FUNCTION_BLOCK FB_EnableAxes
VAR_INPUT
	bEnableAxes			: BOOL;
	fOverride			: LREAL;
END_VAR
VAR_OUTPUT
	bAllAxesReady		: BOOL;
	bActive				: BOOL;
	bError				: BOOL;
END_VAR
VAR_IN_OUT
	stAxis1				: AXIS_REF;
END_VAR
VAR
	fbPower1			:MC_Power;
END_VAR

fbPower1(
	Enable:=bEnableAxes, 
	Enable_Positive:=bEnableAxes, 
	Enable_Negative:=bEnableAxes, 
	Override:=fOverride, 
	BufferMode:= , 
	Axis:=stAxis1, 
	Status=> , 
	Busy=> , 
	Active=> , 
	Error=> , 
	ErrorID=> );

IF fbPower1.Active THEN
	bActive := TRUE;
	IF fbPower1.Error THEN
		bError := TRUE;
	ELSE 
		bAllAxesReady := fbPower1.Status;
		bError := FALSE;
	END_IF
ELSE
	bActive := FALSE;
END_IF

END_FUNCTION_BLOCK

(* stored: Version 1.1.0.1, ProductVersion 3.1.4024.12
   POU FB_EnableAxes: Id {8d38cc83-e6cf-443d-a5a4-82a31e086b6d}, SpecialFunc None *)
